SUBAPPLICATION Zaehler (* Subapplication Type *)
  (* Standard: 61499-2 *)
  (* Version 1.0, 2023-02-17, Franz *)
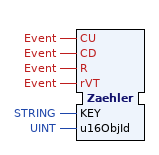
  EVENT_INPUT
    CU; (* Count Up *)
    CD; (* Count Down *)
    R; (* Reset *)
    rVT; (* refresh VT *)
  END_EVENT
  VAR_INPUT
    KEY : STRING;
    u16ObjId : UINT;
  END_VAR
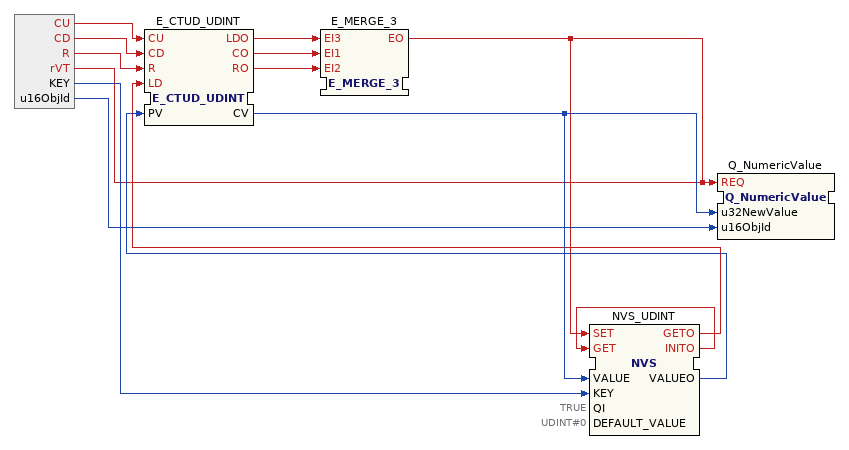
  FBS
    E_CTUD_UDINT : iec61499::events::E_CTUD_UDINT;
    Q_NumericValue : isobus::UT::Q::Q_NumericValue;
    NVS_UDINT : logiBUS::storage::esp32_nvs::NVS(QI := TRUE, DEFAULT_VALUE := UDINT#0);
    E_MERGE_3 : iec61499::events::E_MERGE_3;
  END_FBS
  EVENT_CONNECTIONS
    E_MERGE_3.EO TO Q_NumericValue.REQ;
    CU TO E_CTUD_UDINT.CU;
    CD TO E_CTUD_UDINT.CD;
    R TO E_CTUD_UDINT.R;
    rVT TO Q_NumericValue.REQ;
    E_MERGE_3.EO TO NVS_UDINT.SET;
    NVS_UDINT.GETO TO E_CTUD_UDINT.LD;
    NVS_UDINT.INITO TO NVS_UDINT.GET;
    E_CTUD_UDINT.LDO TO E_MERGE_3.EI3;
    E_CTUD_UDINT.CO TO E_MERGE_3.EI1;
    E_CTUD_UDINT.RO TO E_MERGE_3.EI2;
  END_CONNECTIONS
  DATA_CONNECTIONS
    E_CTUD_UDINT.CV TO Q_NumericValue.u32NewValue;
    u16ObjId TO Q_NumericValue.u16ObjId;
    E_CTUD_UDINT.CV TO NVS_UDINT.VALUE;
    NVS_UDINT.VALUEO TO E_CTUD_UDINT.PV;
    KEY TO NVS_UDINT.KEY;
  END_CONNECTIONS
END_SUBAPPLICATION
